FUNCTION_BLOCK TransportSequenceGoHome EXTENDS TransportSequence IMPLEMENTS ZCore.ISequence
VAR
  _step : ZCore.Step(TransportStep.GohomeBegin, TransportStep.GohomeEnd);
  _timer : ZAux.Timer;
END_VAR

IF NOT Busy THEN
  RETURN;
END_IF

IF OnStart(_step) THEN
  ; // init custom sequence variables here ...
END_IF

IF OnStop() THEN
  RETURN; // external stop was triggered
END_IF

IF OnHalt() THEN
  ; // Halting := TRUE; // Uncomment to acknowledge that the sequence is halting
END_IF

REPEAT
  LogStep();

  CASE _step.Index OF
    (* -------------------------------------------------------------------------------------------------------------------------------- *)
    TransportStep.GoHomeBegin:
    (* -------------------------------------------------------------------------------------------------------------------------------- *)
      IF _step.OnEntry()
      THEN
        _timer.WaitAsync(2);
			END_IF
      
      Await(_timer, nextStep:=TransportStep.GoHomeVerticalUp);

    (* -------------------------------------------------------------------------------------------------------------------------------- *)
    TransportStep.GoHomeVerticalUp:
    (* -------------------------------------------------------------------------------------------------------------------------------- *)
      IF _step.OnEntry()
      THEN        
        _axis.VerticalZ.MoveAbsoluteAsync(startToken:=THIS^, position:=_data.Machine.VerticalHomePos, speed:=_data.Machine.Slowspeed);
      END_IF
      
      Await(obj1:=_axis.VerticalZ, nextStep:=TransportStep.GoHomeHorizontalToRightPos);

    (* -------------------------------------------------------------------------------------------------------------------------------- *)
    TransportStep.GoHomeHorizontalToRightPos:
    (* -------------------------------------------------------------------------------------------------------------------------------- *)
      IF _step.OnEntry()
      THEN        
        _axis.HorizontalX.MoveAbsoluteAsync(startToken:=THIS^, position:=_data.Machine.HorizontalHomePos, speed:=_data.Machine.Slowspeed);
      END_IF
      
      Await(obj1:=_axis.HorizontalX, nextStep:=TransportStep.GoHomeUnlockQualityInspection);

    (* -------------------------------------------------------------------------------------------------------------------------------- *)
    TransportStep.GoHomeUnlockQualityInspection:
    (* -------------------------------------------------------------------------------------------------------------------------------- *)
      _unit.QualityInspection.Unlock(unit:=_parent);
      _step.SetNext(index:=TransportStep.GoHomeStartHomingOfChilds);

    (* -------------------------------------------------------------------------------------------------------------------------------- *)
    TransportStep.GoHomeStartHomingOfChilds:
    (* -------------------------------------------------------------------------------------------------------------------------------- *)
      IF _step.OnEntry()
      THEN        
        _unit.Assembly.HomingAsync(startToken:=THIS^, unit:=0); // <- For homing we do not need to lock, therefore 0 on second parameter)
        _unit.Drilling.HomingAsync(startToken:=THIS^, unit:=0);
        _unit.QualityInspection.HomingAsync(THIS^, 0);
      END_IF
      
      Await3(obj1:=_unit.Assembly, obj2:=_unit.Drilling, obj3:=_unit.QualityInspection, nextStep:=TransportStep.GoHomeEnd);

    (* -------------------------------------------------------------------------------------------------------------------------------- *)
    TransportStep.GoHomeEnd:
    (* -------------------------------------------------------------------------------------------------------------------------------- *)
      SetBusy(FALSE);
  
  ELSE
    Abort('sequence contains unhandled step');
  END_CASE
UNTIL _step.IsNotRepeatable() OR_ELSE NOT Busy END_REPEAT

END_FUNCTION_BLOCK

(* stored: Version 1.1.0.1
   POU TransportSequenceGoHome: Id {0a50907f-f317-41aa-84cc-d85c42ee1443}, SpecialFunc None *)
